SUBAPPLICATION Uebung_002c (* DigitalInput_I1/_I2 auf DigitalOutput_Q1 *)
  (* Standard: 61499-2; Description: Copyright (c) 2023 Meisterschulen am Ostbahnhof This program and the accompanying materials are made available under the terms of the Eclipse Public License 2.0 which is available at https://www.eclipse.org/legal/epl-2.0/ SPDX-License-Identifier: EPL-2.0 *)
  (* Version 1.0, 2023-10-23, Franz Höpfinger, Meisterschulen am Ostbahnhof *)
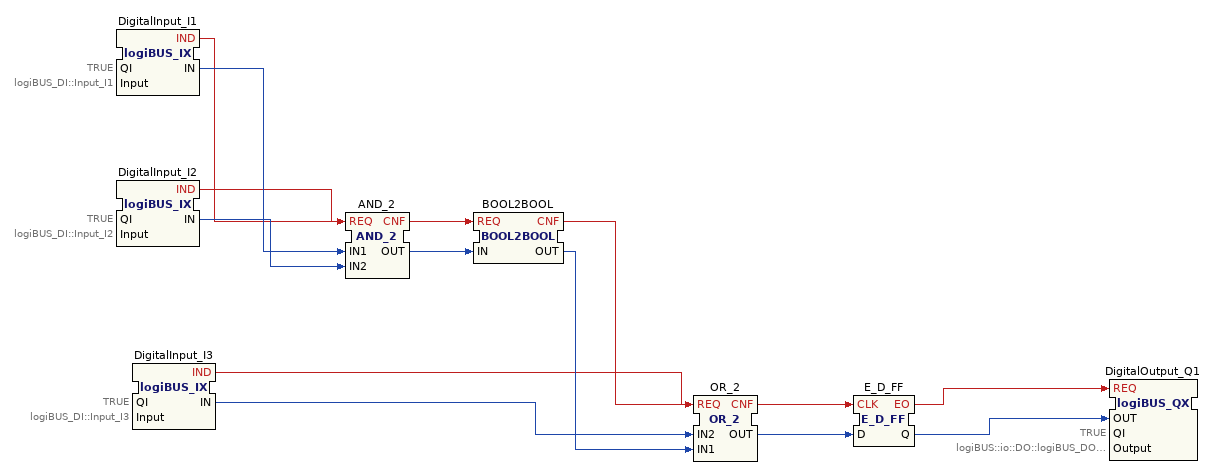
  FBS
    DigitalOutput_Q1 : logiBUS_QX(QI := TRUE, Output := logiBUS::io::DO::logiBUS_DO::Output_Q1);
    DigitalInput_I1 : logiBUS_IX(QI := TRUE, Input := logiBUS_DI::Input_I1);
    DigitalInput_I2 : logiBUS_IX(QI := TRUE, Input := logiBUS_DI::Input_I2);
    AND_2 : AND_2;
    DigitalInput_I3 : logiBUS_IX(QI := TRUE, Input := logiBUS_DI::Input_I3);
    OR_2 : OR_2;
    BOOL2BOOL : BOOL2BOOL;
    E_D_FF : E_D_FF;
  END_FBS
  EVENT_CONNECTIONS
    DigitalInput_I1.IND TO AND_2.REQ;
    DigitalInput_I2.IND TO AND_2.REQ;
    E_D_FF.EO TO DigitalOutput_Q1.REQ;
    AND_2.CNF TO BOOL2BOOL.REQ;
    BOOL2BOOL.CNF TO OR_2.REQ;
    DigitalInput_I3.IND TO OR_2.REQ;
    OR_2.CNF TO E_D_FF.CLK;
  END_CONNECTIONS
  DATA_CONNECTIONS
    DigitalInput_I1.IN TO AND_2.IN1;
    DigitalInput_I2.IN TO AND_2.IN2;
    DigitalInput_I3.IN TO OR_2.IN2;
    E_D_FF.Q TO DigitalOutput_Q1.OUT;
    AND_2.OUT TO BOOL2BOOL.IN;
    BOOL2BOOL.OUT TO OR_2.IN1;
    OR_2.OUT TO E_D_FF.D;
  END_CONNECTIONS
END_SUBAPPLICATION
